(* PLC project Untitled1, Beckhoff Automation GmbH TF6420 Database Server Query Analyser 1.0.0.0 *)
(* stored: creationDateTime 2021-07-21T09:14:47, modificationDateTime 2021-07-21T09:14:47 *)

TYPE DUT_AlarmDB : STRUCT
  id : LINT;
  sName : STRING(255);
  tActiveStartTime : STRING(255);
  tAckTime : STRING(255);
  tClearedTime : STRING(255);
  uiRepeatCount : DINT;
  sAlarmText : STRING(255);
  bIsActive : INT;
  bIsAcknowledged : INT;
END_STRUCT;
END_TYPE
